// SIMATIC STEP 7 (V5.x) project examen2
// CPU: CPU 317-2 DP
// station: Hardware
// station: SIMATIC 300(1)
// station: P_ADR_BUS
// program: S7 Program(1)

SYMBOL_TABLE
"Prueba 1"	FB 1	FB 1
"Prueba 2"	FB 2	FB 2
"Prueba 3"	FB 3	FB 3
"Prueba 4"	FB 4	FB 4
"Prueba 5"	FB 5	FB 5
"Prueba 6"	FB 6	FB 6
"Prueba 8"	FB 8	FB 8
"Prueba 9"	FB 9	FB 9
"1HONGO"	I 0.0	BOOL
"1RESET"	I 0.1	BOOL
"1LOCAL"	I 0.2	BOOL
"1REMOTO"	I 0.3	BOOL
"1C_UNICO"	I 0.4	BOOL
"1C_CONTINUO"	I 0.5	BOOL
"1PARO"	I 0.6	BOOL
"1A0"	I 1.0	BOOL
"1A1"	I 1.1	BOOL
"1B0"	I 1.2	BOOL
"1B1"	I 1.3	BOOL
"2HONGO"	I 2.0	BOOL
"2RESET"	I 2.1	BOOL
"2LOCAL"	I 2.2	BOOL
"2REMOTO"	I 2.3	BOOL
"2C_UNICO"	I 2.4	BOOL
"2C_CONTINUO"	I 2.5	BOOL
"2PARO"	I 2.6	BOOL
"2A0"	I 3.0	BOOL
"2A1"	I 3.1	BOOL
"2B0"	I 3.2	BOOL
"2B1"	I 3.3	BOOL
"3HONGO"	I 4.0	BOOL
"3RESET"	I 4.1	BOOL
"3LOCAL"	I 4.2	BOOL
"3REMOTO"	I 4.3	BOOL
"3C_UNICO"	I 4.4	BOOL
"3C_CONTINUO"	I 4.5	BOOL
"3PARO"	I 4.6	BOOL
"3A0"	I 5.0	BOOL
"3A1"	I 5.1	BOOL
"3B0"	I 5.2	BOOL
"3B1"	I 5.3	BOOL
"3C0"	I 5.4	BOOL
"3C1"	I 5.5	BOOL
"4HONGO"	I 6.0	BOOL
"4RESET"	I 6.1	BOOL
"4LOCAL"	I 6.2	BOOL
"4REMOTO"	I 6.3	BOOL
"4C_UNICO"	I 6.4	BOOL
"4C_CONTINUO"	I 6.5	BOOL
"4PARO"	I 6.6	BOOL
"4C2"	I 6.7	BOOL
"4A0"	I 7.0	BOOL
"4A1"	I 7.1	BOOL
"4B0"	I 7.2	BOOL
"4B1"	I 7.3	BOOL
"4C0"	I 7.4	BOOL
"4C1"	I 7.5	BOOL
"4D0"	I 7.6	BOOL
"4D1"	I 7.7	BOOL
"5HONGO"	I 8.0	BOOL
"5RESET"	I 8.1	BOOL
"5LOCAL"	I 8.2	BOOL
"5REMOTO"	I 8.3	BOOL
"5C_UNICO"	I 8.4	BOOL
"5C_CONTINUO"	I 8.5	BOOL
"5PARO"	I 8.6	BOOL
"5A0"	I 9.0	BOOL
"5A1"	I 9.1	BOOL
"5B0"	I 9.2	BOOL
"5B1"	I 9.3	BOOL
"5C0"	I 9.4	BOOL
"5C1"	I 9.5	BOOL
"6HONGO"	I 10.0	BOOL
"6RESET"	I 10.1	BOOL
"6LOCAL"	I 10.2	BOOL
"6REMOTO"	I 10.3	BOOL
"6C_UNICO"	I 10.4	BOOL
"6C_CONTINUO"	I 10.5	BOOL
"6PARO"	I 10.6	BOOL
"6A0"	I 11.0	BOOL
"6A1"	I 11.1	BOOL
"6B0"	I 11.2	BOOL
"6B1"	I 11.3	BOOL
"6C0"	I 11.4	BOOL
"6C1"	I 11.5	BOOL
"6D0"	I 11.6	BOOL
"6D1"	I 11.7	BOOL
"8HONGO"	I 12.0	BOOL
"8RESET"	I 12.1	BOOL
"8LOCAL"	I 12.2	BOOL
"8REMOTO"	I 12.3	BOOL
"8C_UNICO"	I 12.4	BOOL
"8C_CONTINUO"	I 12.5	BOOL
"8PARO"	I 12.6	BOOL
"8A0"	I 13.0	BOOL
"8A1"	I 13.1	BOOL
"8B0"	I 13.2	BOOL
"8B1"	I 13.3	BOOL
"8C0"	I 13.4	BOOL
"8C1"	I 13.5	BOOL
"9HONGO"	I 14.0	BOOL
"9RESET"	I 14.1	BOOL
"9LOCAL"	I 14.2	BOOL
"9REMOTO"	I 14.3	BOOL
"9C_UNICO"	I 14.4	BOOL
"9C_CONTINUO"	I 14.5	BOOL
"9PARO"	I 14.6	BOOL
"9A1"	I 15.0	BOOL
"9A2"	I 15.1	BOOL
"9A3"	I 15.2	BOOL
"1Y1"	Q 0.0	BOOL
"1Y2"	Q 0.1	BOOL
"1Y3"	Q 0.2	BOOL
"1Y4"	Q 0.3	BOOL
"2Y1"	Q 1.0	BOOL
"2Y2"	Q 1.1	BOOL
"2Y3"	Q 1.2	BOOL
"2Y4"	Q 1.3	BOOL
"3Y1"	Q 2.0	BOOL
"3Y2"	Q 2.1	BOOL
"3Y3"	Q 2.2	BOOL
"3Y4"	Q 2.3	BOOL
"3Y5"	Q 2.4	BOOL
"3Y6"	Q 2.5	BOOL
"4Y1"	Q 3.0	BOOL
"4Y2"	Q 3.1	BOOL
"4Y3"	Q 3.2	BOOL
"4Y4"	Q 3.3	BOOL
"4Y5"	Q 3.4	BOOL
"4Y6"	Q 3.5	BOOL
"4Y7"	Q 3.6	BOOL
"4Y8"	Q 3.7	BOOL
"5Y1"	Q 4.0	BOOL
"5Y2"	Q 4.1	BOOL
"5Y3"	Q 4.2	BOOL
"5Y4"	Q 4.3	BOOL
"5Y5"	Q 4.4	BOOL
"5Y6"	Q 4.5	BOOL
"6Y1"	Q 5.0	BOOL
"6Y2"	Q 5.1	BOOL
"6Y3"	Q 5.2	BOOL
"6Y4"	Q 5.3	BOOL
"6Y5"	Q 5.4	BOOL
"6Y6"	Q 5.5	BOOL
"6Y7"	Q 5.6	BOOL
"6Y8"	Q 5.7	BOOL
"8Y1"	Q 6.0	BOOL
"8Y2"	Q 6.1	BOOL
"8Y3"	Q 6.2	BOOL
"8Y4"	Q 6.3	BOOL
"8Y5"	Q 6.4	BOOL
"8Y6"	Q 6.5	BOOL
"9Y1"	Q 7.0	BOOL
"9Y2"	Q 7.1	BOOL
END_SYMBOL_TABLE

FUNCTION_BLOCK "Prueba 1"	// FB 1
VERSION : 0.1
VAR
  K1 : BOOL ;
  KA : BOOL ;
  KB : BOOL ;
  K0 : BOOL ;
  K2 : BOOL ;
  K3 : BOOL ;
  K4 : BOOL ;
  K5 : BOOL ;
  K6 : BOOL ;
  K7 : BOOL ;
  K8 : BOOL ;
  KT8 : BOOL ;
  K9 : BOOL ;
END_VAR
BEGIN
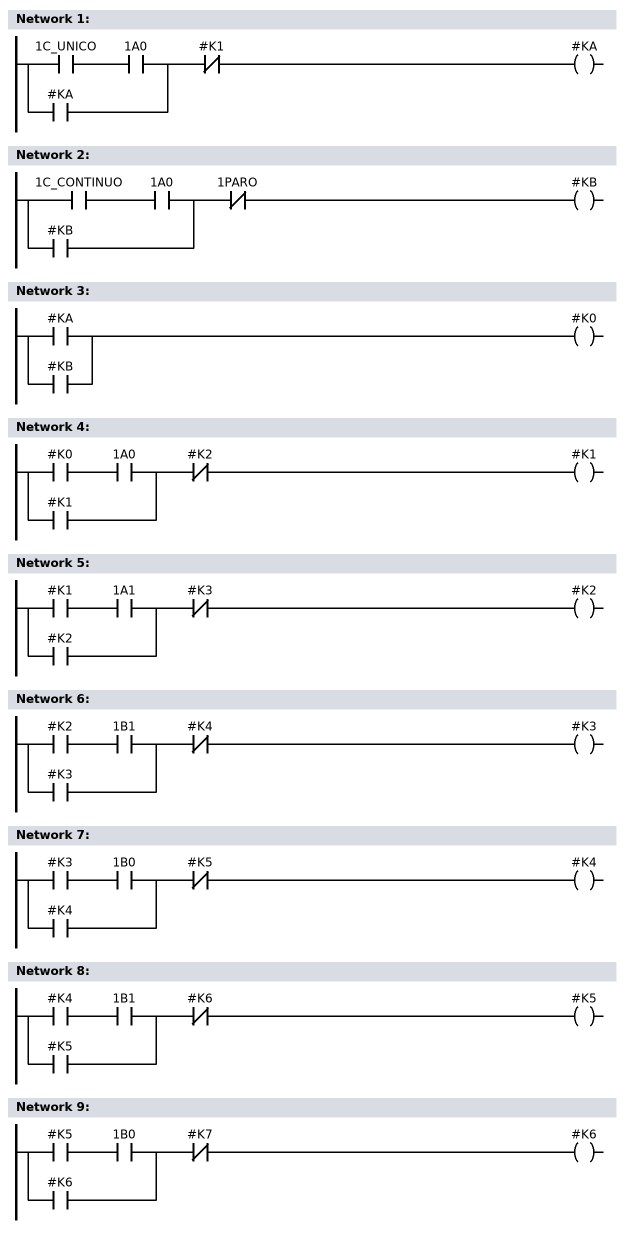
NETWORK
TITLE =
      A(;
      A     "1C_UNICO";
      A     "1A0";
      O     #KA;
      );
      AN    #K1;
      =     #KA;
NETWORK
TITLE =
      A(;
      A     "1C_CONTINUO";
      A     "1A0";
      O     #KB;
      );
      AN    "1PARO";
      =     #KB;
NETWORK
TITLE =
      O     #KA;
      O     #KB;
      =     #K0;
NETWORK
TITLE =
      A(;
      A     #K0;
      A     "1A0";
      O     #K1;
      );
      AN    #K2;
      =     #K1;
NETWORK
TITLE =
      A(;
      A     #K1;
      A     "1A1";
      O     #K2;
      );
      AN    #K3;
      =     #K2;
NETWORK
TITLE =
      A(;
      A     #K2;
      A     "1B1";
      O     #K3;
      );
      AN    #K4;
      =     #K3;
NETWORK
TITLE =
      A(;
      A     #K3;
      A     "1B0";
      O     #K4;
      );
      AN    #K5;
      =     #K4;
NETWORK
TITLE =
      A(;
      A     #K4;
      A     "1B1";
      O     #K5;
      );
      AN    #K6;
      =     #K5;
NETWORK
TITLE =
      A(;
      A     #K5;
      A     "1B0";
      O     #K6;
      );
      AN    #K7;
      =     #K6;
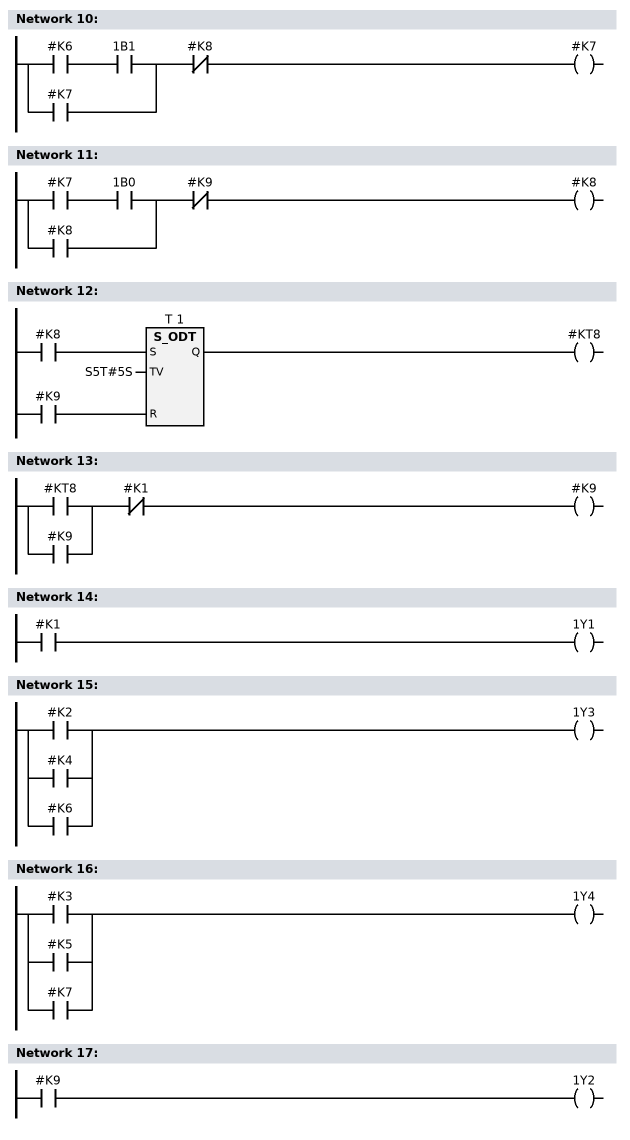
NETWORK
TITLE =
      A(;
      A     #K6;
      A     "1B1";
      O     #K7;
      );
      AN    #K8;
      =     #K7;
NETWORK
TITLE =
      A(;
      A     #K7;
      A     "1B0";
      O     #K8;
      );
      AN    #K9;
      =     #K8;
NETWORK
TITLE =
      A     #K8;
      L     S5T#5S;
      SD    T 1;
      A     #K9;
      R     T 1;
      NOP   0;
      NOP   0;
      A     T 1;
      =     #KT8;
NETWORK
TITLE =
      A(;
      O     #KT8;
      O     #K9;
      );
      AN    #K1;
      =     #K9;
NETWORK
TITLE =
      A     #K1;
      =     "1Y1";
NETWORK
TITLE =
      O     #K2;
      O     #K4;
      O     #K6;
      =     "1Y3";
NETWORK
TITLE =
      O     #K3;
      O     #K5;
      O     #K7;
      =     "1Y4";
NETWORK
TITLE =
      A     #K9;
      =     "1Y2";
END_FUNCTION_BLOCK

FUNCTION_BLOCK "Prueba 2"	// FB 2
VERSION : 0.1
VAR
  K0 : BOOL ;
  K1 : BOOL ;
  K2 : BOOL ;
  K3 : BOOL ;
  K4 : BOOL ;
  K5 : BOOL ;
  K6 : BOOL ;
  K7 : BOOL ;
  K8 : BOOL ;
  KT : BOOL ;
  KA : BOOL ;
  KB : BOOL ;
  kt2 : BOOL ;
END_VAR
BEGIN
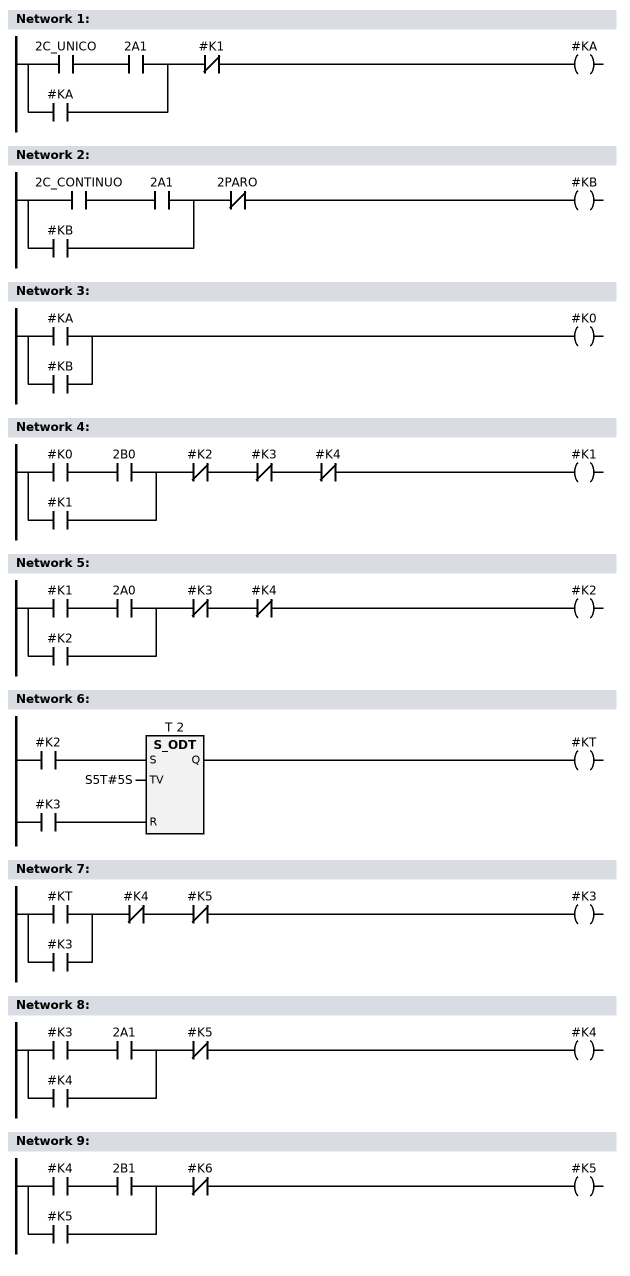
NETWORK
TITLE =
      A(;
      A     "2C_UNICO";
      A     "2A1";
      O     #KA;
      );
      AN    #K1;
      =     #KA;
NETWORK
TITLE =
      A(;
      A     "2C_CONTINUO";
      A     "2A1";
      O     #KB;
      );
      AN    "2PARO";
      =     #KB;
NETWORK
TITLE =
      O     #KA;
      O     #KB;
      =     #K0;
NETWORK
TITLE =
      A(;
      A     #K0;
      A     "2B0";
      O     #K1;
      );
      AN    #K2;
      AN    #K3;
      AN    #K4;
      =     #K1;
NETWORK
TITLE =
      A(;
      A     #K1;
      A     "2A0";
      O     #K2;
      );
      AN    #K3;
      AN    #K4;
      =     #K2;
NETWORK
TITLE =
      A     #K2;
      L     S5T#5S;
      SD    T 2;
      A     #K3;
      R     T 2;
      NOP   0;
      NOP   0;
      A     T 2;
      =     #KT;
NETWORK
TITLE =
      A(;
      O     #KT;
      O     #K3;
      );
      AN    #K4;
      AN    #K5;
      =     #K3;
NETWORK
TITLE =
      A(;
      A     #K3;
      A     "2A1";
      O     #K4;
      );
      AN    #K5;
      =     #K4;
NETWORK
TITLE =
      A(;
      A     #K4;
      A     "2B1";
      O     #K5;
      );
      AN    #K6;
      =     #K5;
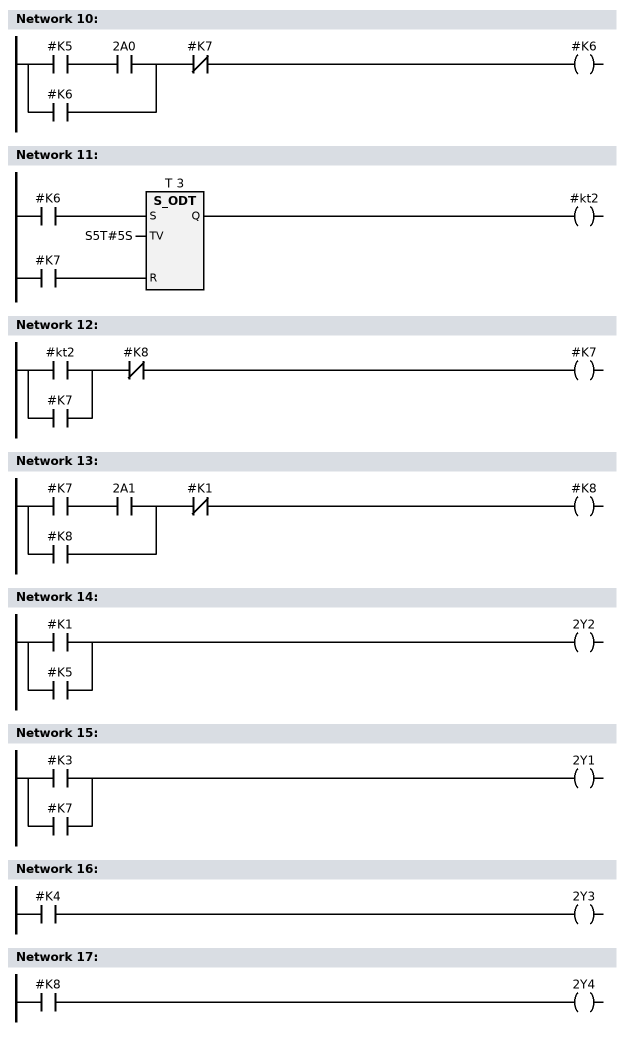
NETWORK
TITLE =
      A(;
      A     #K5;
      A     "2A0";
      O     #K6;
      );
      AN    #K7;
      =     #K6;
NETWORK
TITLE =
      A     #K6;
      L     S5T#5S;
      SD    T 3;
      A     #K7;
      R     T 3;
      NOP   0;
      NOP   0;
      A     T 3;
      =     #kt2;
NETWORK
TITLE =
      A(;
      O     #kt2;
      O     #K7;
      );
      AN    #K8;
      =     #K7;
NETWORK
TITLE =
      A(;
      A     #K7;
      A     "2A1";
      O     #K8;
      );
      AN    #K1;
      =     #K8;
NETWORK
TITLE =
      O     #K1;
      O     #K5;
      =     "2Y2";
NETWORK
TITLE =
      O     #K3;
      O     #K7;
      =     "2Y1";
NETWORK
TITLE =
      A     #K4;
      =     "2Y3";
NETWORK
TITLE =
      A     #K8;
      =     "2Y4";
END_FUNCTION_BLOCK

FUNCTION_BLOCK "Prueba 3"	// FB 3
VERSION : 0.1
VAR
  KA : BOOL ;
  KB : BOOL ;
  K0 : BOOL ;
  K1 : BOOL ;
  K2 : BOOL ;
  K3 : BOOL ;
  K4 : BOOL ;
  K5 : BOOL ;
  K6 : BOOL ;
  K7 : BOOL ;
END_VAR
BEGIN
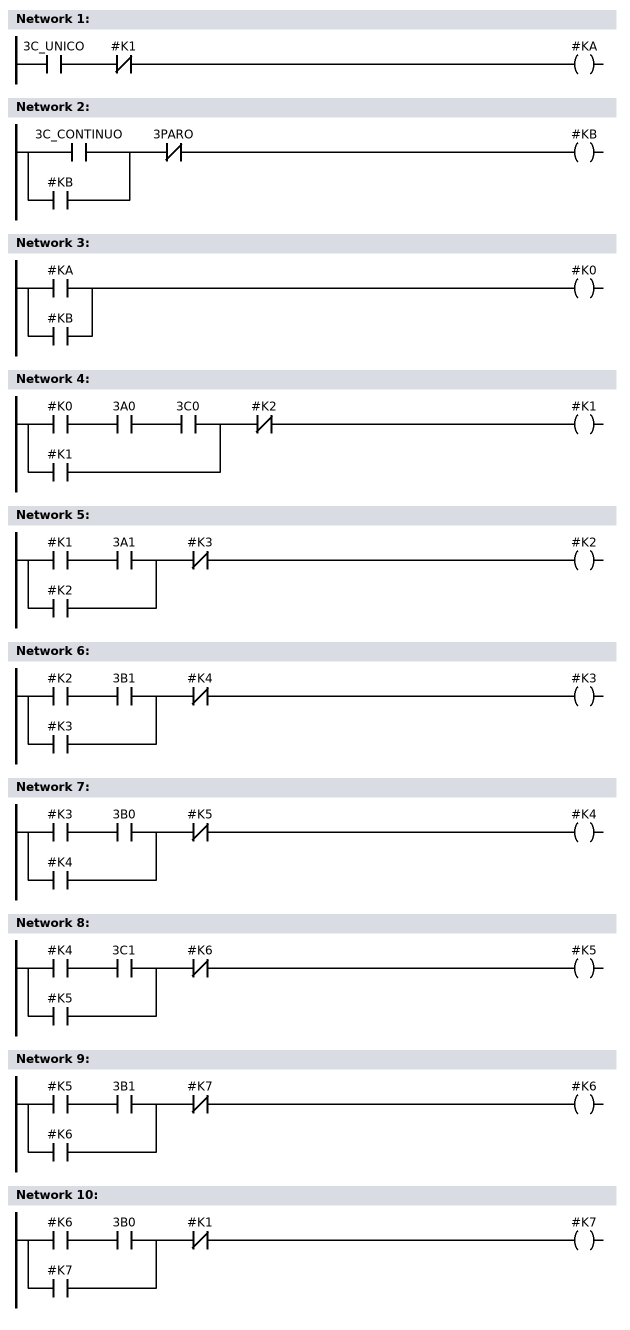
NETWORK
TITLE =
      A     "3C_UNICO";
      AN    #K1;
      =     #KA;
NETWORK
TITLE =
      A(;
      O     "3C_CONTINUO";
      O     #KB;
      );
      AN    "3PARO";
      =     #KB;
NETWORK
TITLE =
      O     #KA;
      O     #KB;
      =     #K0;
NETWORK
TITLE =
      A(;
      A     #K0;
      A     "3A0";
      A     "3C0";
      O     #K1;
      );
      AN    #K2;
      =     #K1;
NETWORK
TITLE =
      A(;
      A     #K1;
      A     "3A1";
      O     #K2;
      );
      AN    #K3;
      =     #K2;
NETWORK
TITLE =
      A(;
      A     #K2;
      A     "3B1";
      O     #K3;
      );
      AN    #K4;
      =     #K3;
NETWORK
TITLE =
      A(;
      A     #K3;
      A     "3B0";
      O     #K4;
      );
      AN    #K5;
      =     #K4;
NETWORK
TITLE =
      A(;
      A     #K4;
      A     "3C1";
      O     #K5;
      );
      AN    #K6;
      =     #K5;
NETWORK
TITLE =
      A(;
      A     #K5;
      A     "3B1";
      O     #K6;
      );
      AN    #K7;
      =     #K6;
NETWORK
TITLE =
      A(;
      A     #K6;
      A     "3B0";
      O     #K7;
      );
      AN    #K1;
      =     #K7;
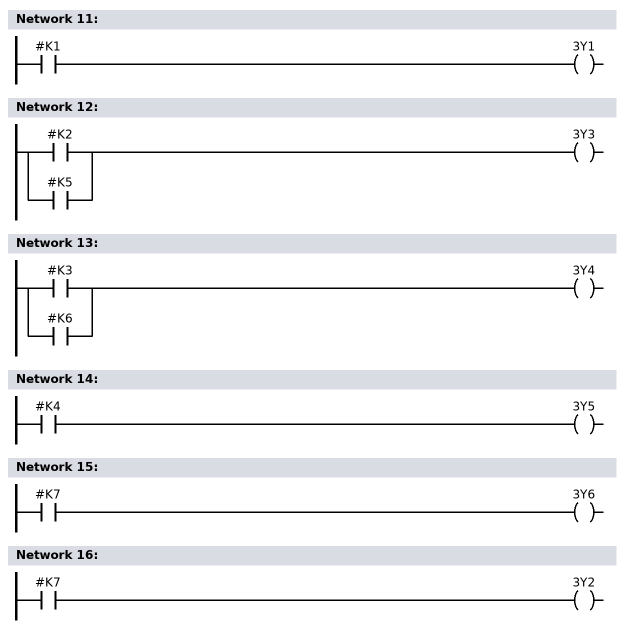
NETWORK
TITLE =
      A     #K1;
      =     "3Y1";
NETWORK
TITLE =
      O     #K2;
      O     #K5;
      =     "3Y3";
NETWORK
TITLE =
      O     #K3;
      O     #K6;
      =     "3Y4";
NETWORK
TITLE =
      A     #K4;
      =     "3Y5";
NETWORK
TITLE =
      A     #K7;
      =     "3Y6";
NETWORK
TITLE =
      A     #K7;
      =     "3Y2";
END_FUNCTION_BLOCK

FUNCTION_BLOCK "Prueba 4"	// FB 4
TITLE = Prueba 4
VERSION : 0.1
VAR
  KA : BOOL ;
  KB : BOOL ;
  K0 : BOOL ;
  K1 : BOOL ;
  K2 : BOOL ;
  K3 : BOOL ;
  K4 : BOOL ;
  K5 : BOOL ;
  K6 : BOOL ;
  K7 : BOOL ;
  K8 : BOOL ;
  K9 : BOOL ;
  KT : BOOL ;
END_VAR
BEGIN
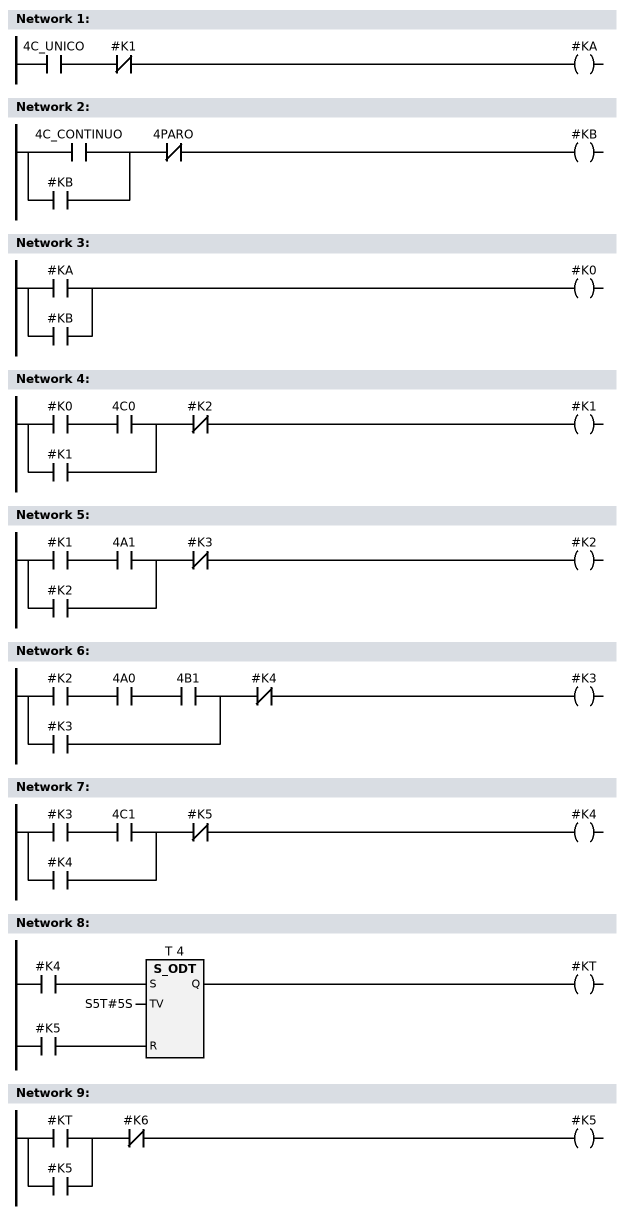
NETWORK
TITLE =
      A     "4C_UNICO";
      AN    #K1;
      =     #KA;
NETWORK
TITLE =
      A(;
      O     "4C_CONTINUO";
      O     #KB;
      );
      AN    "4PARO";
      =     #KB;
NETWORK
TITLE =
      O     #KA;
      O     #KB;
      =     #K0;
NETWORK
TITLE =
      A(;
      A     #K0;
      A     "4C0";
      O     #K1;
      );
      AN    #K2;
      =     #K1;
NETWORK
TITLE =
      A(;
      A     #K1;
      A     "4A1";
      O     #K2;
      );
      AN    #K3;
      =     #K2;
NETWORK
TITLE =
      A(;
      A     #K2;
      A     "4A0";
      A     "4B1";
      O     #K3;
      );
      AN    #K4;
      =     #K3;
NETWORK
TITLE =
      A(;
      A     #K3;
      A     "4C1";
      O     #K4;
      );
      AN    #K5;
      =     #K4;
NETWORK
TITLE =
      A     #K4;
      L     S5T#5S;
      SD    T 4;
      A     #K5;
      R     T 4;
      NOP   0;
      NOP   0;
      A     T 4;
      =     #KT;
NETWORK
TITLE =
      A(;
      O     #KT;
      O     #K5;
      );
      AN    #K6;
      =     #K5;
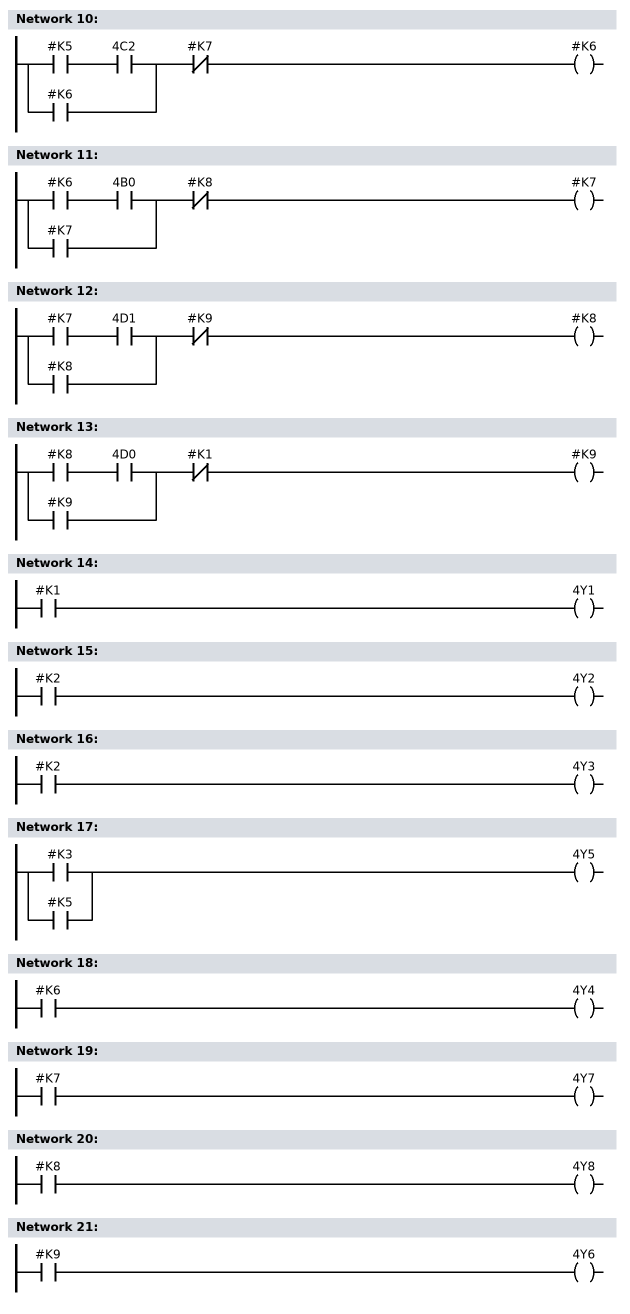
NETWORK
TITLE =
      A(;
      A     #K5;
      A     "4C2";
      O     #K6;
      );
      AN    #K7;
      =     #K6;
NETWORK
TITLE =
      A(;
      A     #K6;
      A     "4B0";
      O     #K7;
      );
      AN    #K8;
      =     #K7;
NETWORK
TITLE =
      A(;
      A     #K7;
      A     "4D1";
      O     #K8;
      );
      AN    #K9;
      =     #K8;
NETWORK
TITLE =
      A(;
      A     #K8;
      A     "4D0";
      O     #K9;
      );
      AN    #K1;
      =     #K9;
NETWORK
TITLE =
      A     #K1;
      =     "4Y1";
NETWORK
TITLE =
      A     #K2;
      =     "4Y2";
NETWORK
TITLE =
      A     #K2;
      =     "4Y3";
NETWORK
TITLE =
      O     #K3;
      O     #K5;
      =     "4Y5";
NETWORK
TITLE =
      A     #K6;
      =     "4Y4";
NETWORK
TITLE =
      A     #K7;
      =     "4Y7";
NETWORK
TITLE =
      A     #K8;
      =     "4Y8";
NETWORK
TITLE =
      A     #K9;
      =     "4Y6";
END_FUNCTION_BLOCK

FUNCTION_BLOCK "Prueba 5"	// FB 5
VERSION : 0.1
VAR
  KA : BOOL ;
  KB : BOOL ;
  K0 : BOOL ;
  K1 : BOOL ;
  K2 : BOOL ;
  K3 : BOOL ;
  K4 : BOOL ;
  K5 : BOOL ;
  K6 : BOOL ;
  K7 : BOOL ;
  K8 : BOOL ;
  K9 : BOOL ;
END_VAR
BEGIN
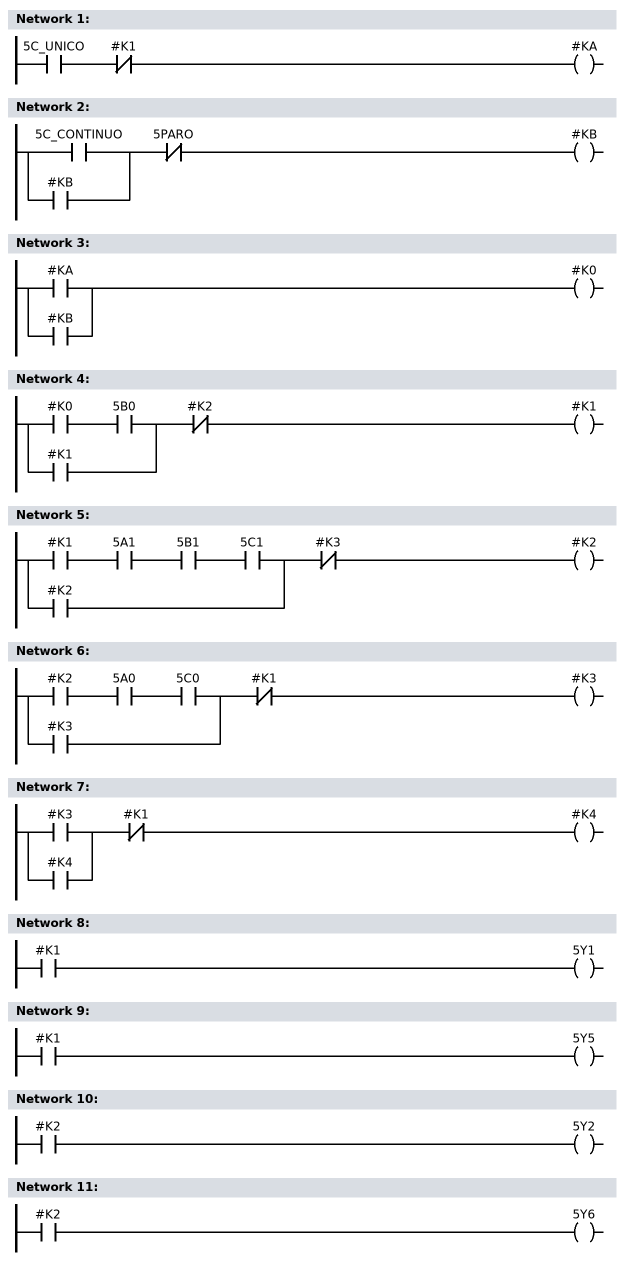
NETWORK
TITLE =
      A     "5C_UNICO";
      AN    #K1;
      =     #KA;
NETWORK
TITLE =
      A(;
      O     "5C_CONTINUO";
      O     #KB;
      );
      AN    "5PARO";
      =     #KB;
NETWORK
TITLE =
      O     #KA;
      O     #KB;
      =     #K0;
NETWORK
TITLE =
      A(;
      A     #K0;
      A     "5B0";
      O     #K1;
      );
      AN    #K2;
      =     #K1;
NETWORK
TITLE =
      A(;
      A     #K1;
      A     "5A1";
      A     "5B1";
      A     "5C1";
      O     #K2;
      );
      AN    #K3;
      =     #K2;
NETWORK
TITLE =
      A(;
      A     #K2;
      A     "5A0";
      A     "5C0";
      O     #K3;
      );
      AN    #K1;
      =     #K3;
NETWORK
TITLE =
      A(;
      O     #K3;
      O     #K4;
      );
      AN    #K1;
      =     #K4;
NETWORK
TITLE =
      A     #K1;
      =     "5Y1";
NETWORK
TITLE =
      A     #K1;
      =     "5Y5";
NETWORK
TITLE =
      A     #K2;
      =     "5Y2";
NETWORK
TITLE =
      A     #K2;
      =     "5Y6";
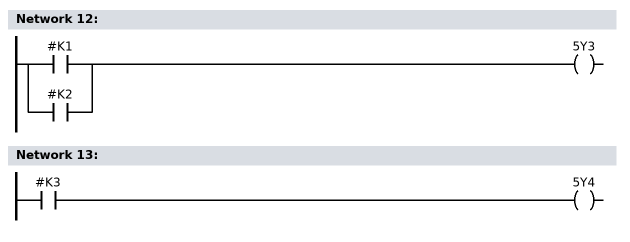
NETWORK
TITLE =
      O     #K1;
      O     #K2;
      =     "5Y3";
NETWORK
TITLE =
      A     #K3;
      =     "5Y4";
END_FUNCTION_BLOCK

FUNCTION_BLOCK "Prueba 6"	// FB 6
VERSION : 0.1
VAR
  KA : BOOL ;
  KB : BOOL ;
  K0 : BOOL ;
  K1 : BOOL ;
  K2 : BOOL ;
  K3 : BOOL ;
  K4 : BOOL ;
  K5 : BOOL ;
  K6 : BOOL ;
  K7 : BOOL ;
  K8 : BOOL ;
  K9 : BOOL ;
END_VAR
BEGIN
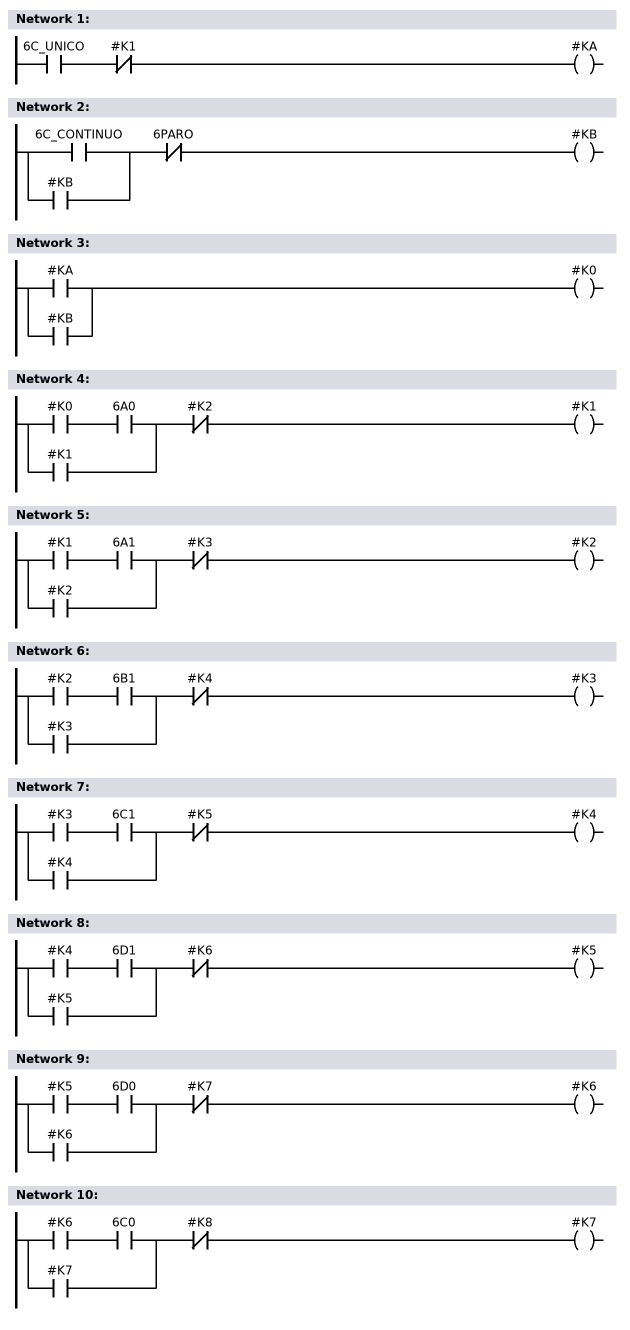
NETWORK
TITLE =
      A     "6C_UNICO";
      AN    #K1;
      =     #KA;
NETWORK
TITLE =
      A(;
      O     "6C_CONTINUO";
      O     #KB;
      );
      AN    "6PARO";
      =     #KB;
NETWORK
TITLE =
      O     #KA;
      O     #KB;
      =     #K0;
NETWORK
TITLE =
      A(;
      A     #K0;
      A     "6A0";
      O     #K1;
      );
      AN    #K2;
      =     #K1;
NETWORK
TITLE =
      A(;
      A     #K1;
      A     "6A1";
      O     #K2;
      );
      AN    #K3;
      =     #K2;
NETWORK
TITLE =
      A(;
      A     #K2;
      A     "6B1";
      O     #K3;
      );
      AN    #K4;
      =     #K3;
NETWORK
TITLE =
      A(;
      A     #K3;
      A     "6C1";
      O     #K4;
      );
      AN    #K5;
      =     #K4;
NETWORK
TITLE =
      A(;
      A     #K4;
      A     "6D1";
      O     #K5;
      );
      AN    #K6;
      =     #K5;
NETWORK
TITLE =
      A(;
      A     #K5;
      A     "6D0";
      O     #K6;
      );
      AN    #K7;
      =     #K6;
NETWORK
TITLE =
      A(;
      A     #K6;
      A     "6C0";
      O     #K7;
      );
      AN    #K8;
      =     #K7;
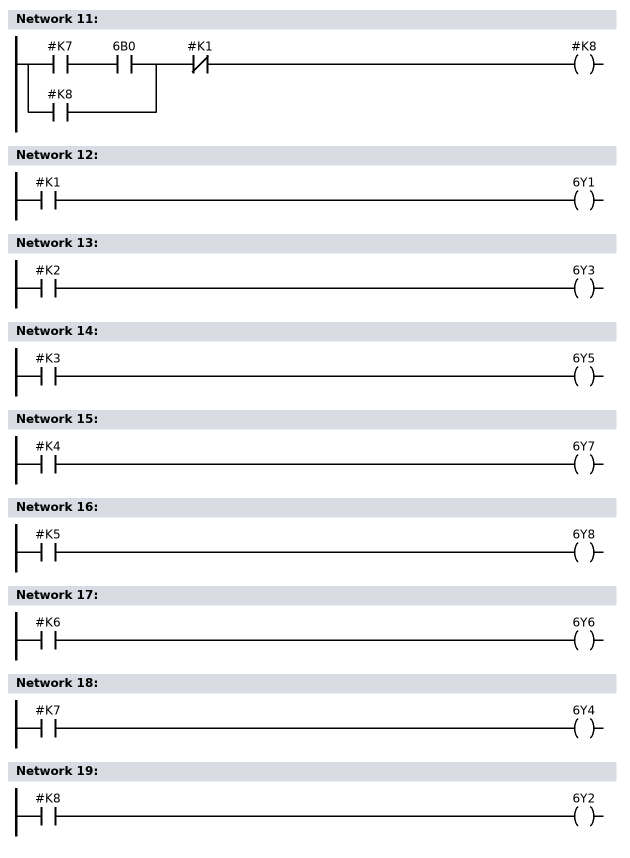
NETWORK
TITLE =
      A(;
      A     #K7;
      A     "6B0";
      O     #K8;
      );
      AN    #K1;
      =     #K8;
NETWORK
TITLE =
      A     #K1;
      =     "6Y1";
NETWORK
TITLE =
      A     #K2;
      =     "6Y3";
NETWORK
TITLE =
      A     #K3;
      =     "6Y5";
NETWORK
TITLE =
      A     #K4;
      =     "6Y7";
NETWORK
TITLE =
      A     #K5;
      =     "6Y8";
NETWORK
TITLE =
      A     #K6;
      =     "6Y6";
NETWORK
TITLE =
      A     #K7;
      =     "6Y4";
NETWORK
TITLE =
      A     #K8;
      =     "6Y2";
END_FUNCTION_BLOCK

FUNCTION_BLOCK "Prueba 8"	// FB 8
VERSION : 0.1
VAR
  KA : BOOL ;
  KB : BOOL ;
  K0 : BOOL ;
  K1 : BOOL ;
  K2 : BOOL ;
  K3 : BOOL ;
  K4 : BOOL ;
  K5 : BOOL ;
  K6 : BOOL ;
  K7 : BOOL ;
  K8 : BOOL ;
  K9 : BOOL ;
END_VAR
BEGIN
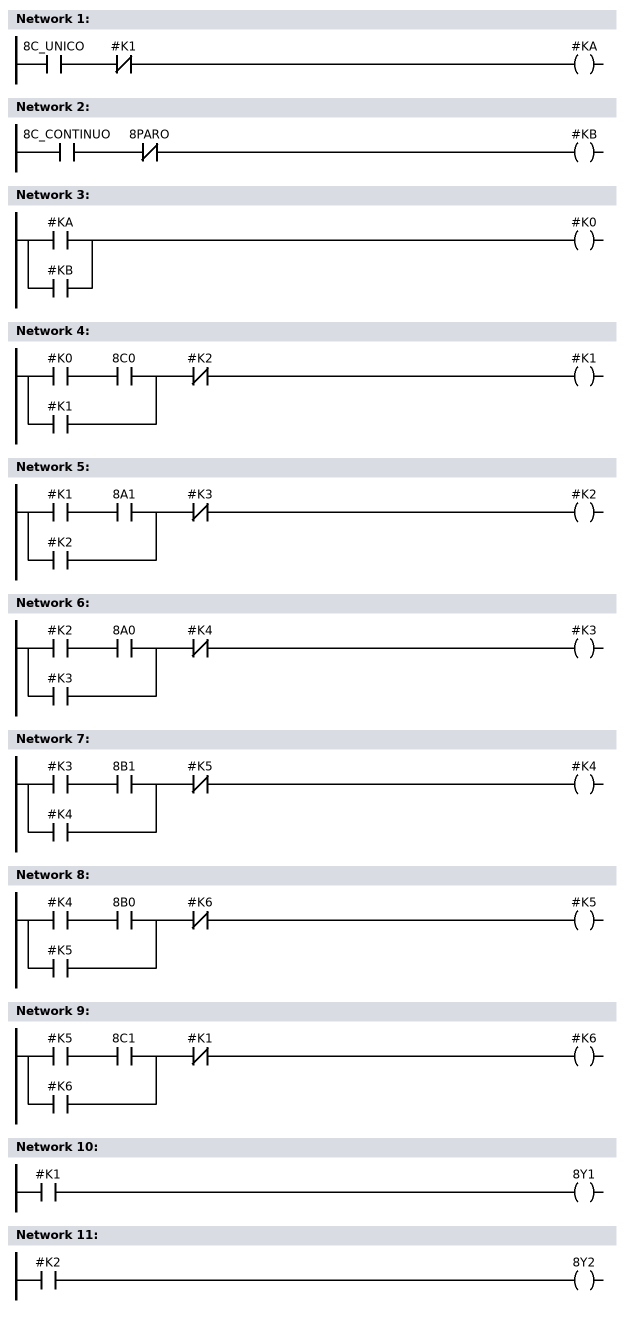
NETWORK
TITLE =
      A     "8C_UNICO";
      AN    #K1;
      =     #KA;
NETWORK
TITLE =
      A     "8C_CONTINUO";
      AN    "8PARO";
      =     #KB;
NETWORK
TITLE =
      O     #KA;
      O     #KB;
      =     #K0;
NETWORK
TITLE =
      A(;
      A     #K0;
      A     "8C0";
      O     #K1;
      );
      AN    #K2;
      =     #K1;
NETWORK
TITLE =
      A(;
      A     #K1;
      A     "8A1";
      O     #K2;
      );
      AN    #K3;
      =     #K2;
NETWORK
TITLE =
      A(;
      A     #K2;
      A     "8A0";
      O     #K3;
      );
      AN    #K4;
      =     #K3;
NETWORK
TITLE =
      A(;
      A     #K3;
      A     "8B1";
      O     #K4;
      );
      AN    #K5;
      =     #K4;
NETWORK
TITLE =
      A(;
      A     #K4;
      A     "8B0";
      O     #K5;
      );
      AN    #K6;
      =     #K5;
NETWORK
TITLE =
      A(;
      A     #K5;
      A     "8C1";
      O     #K6;
      );
      AN    #K1;
      =     #K6;
NETWORK
TITLE =
      A     #K1;
      =     "8Y1";
NETWORK
TITLE =
      A     #K2;
      =     "8Y2";
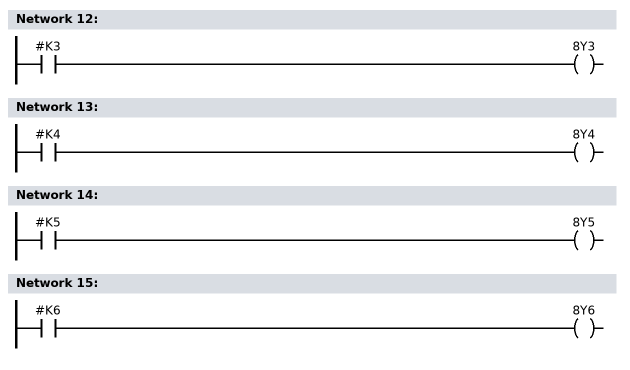
NETWORK
TITLE =
      A     #K3;
      =     "8Y3";
NETWORK
TITLE =
      A     #K4;
      =     "8Y4";
NETWORK
TITLE =
      A     #K5;
      =     "8Y5";
NETWORK
TITLE =
      A     #K6;
      =     "8Y6";
END_FUNCTION_BLOCK

FUNCTION_BLOCK "Prueba 9"	// FB 9
VERSION : 0.1
VAR
  KA : BOOL ;
  KB : BOOL ;
  K0 : BOOL ;
  K1 : BOOL ;
  K2 : BOOL ;
  K3 : BOOL ;
  K4 : BOOL ;
END_VAR
BEGIN
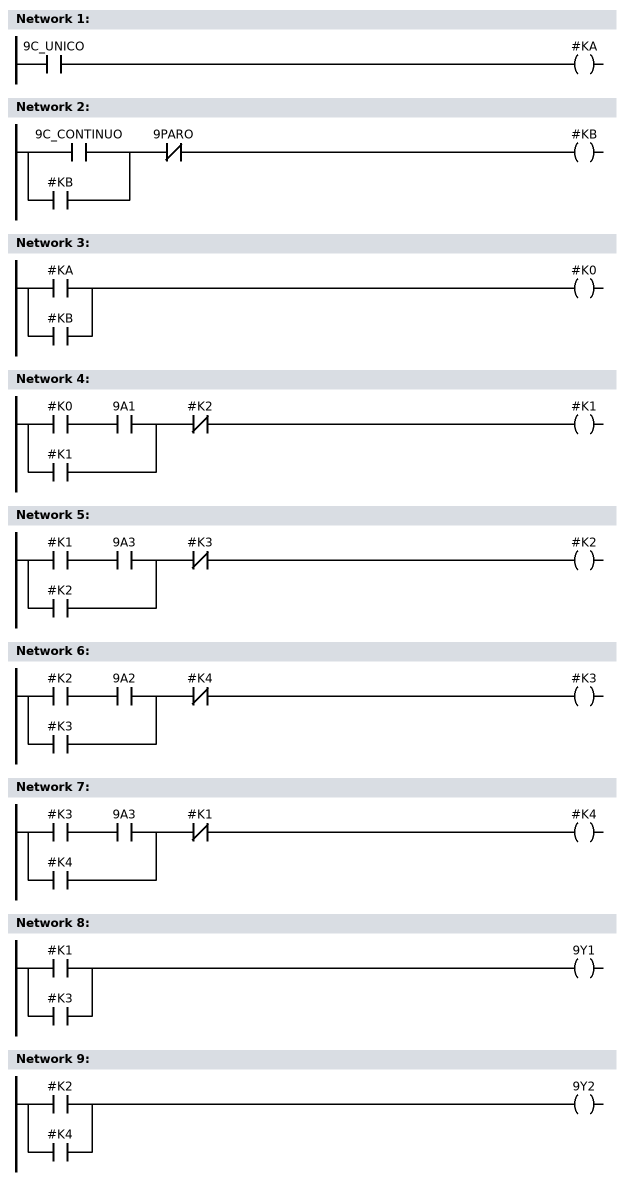
NETWORK
TITLE =
      A     "9C_UNICO";
      =     #KA;
NETWORK
TITLE =
      A(;
      O     "9C_CONTINUO";
      O     #KB;
      );
      AN    "9PARO";
      =     #KB;
NETWORK
TITLE =
      O     #KA;
      O     #KB;
      =     #K0;
NETWORK
TITLE =
      A(;
      A     #K0;
      A     "9A1";
      O     #K1;
      );
      AN    #K2;
      =     #K1;
NETWORK
TITLE =
      A(;
      A     #K1;
      A     "9A3";
      O     #K2;
      );
      AN    #K3;
      =     #K2;
NETWORK
TITLE =
      A(;
      A     #K2;
      A     "9A2";
      O     #K3;
      );
      AN    #K4;
      =     #K3;
NETWORK
TITLE =
      A(;
      A     #K3;
      A     "9A3";
      O     #K4;
      );
      AN    #K1;
      =     #K4;
NETWORK
TITLE =
      O     #K1;
      O     #K3;
      =     "9Y1";
NETWORK
TITLE =
      O     #K2;
      O     #K4;
      =     "9Y2";
END_FUNCTION_BLOCK

DATA_BLOCK DB 1
VERSION : 0.0
"Prueba 1"
BEGIN
END_DATA_BLOCK

DATA_BLOCK DB 2
VERSION : 0.0
"Prueba 2"
BEGIN
END_DATA_BLOCK

DATA_BLOCK DB 3
VERSION : 0.0
"Prueba 3"
BEGIN
END_DATA_BLOCK

DATA_BLOCK DB 4
VERSION : 0.0
"Prueba 4"
BEGIN
END_DATA_BLOCK

DATA_BLOCK DB 5
VERSION : 0.0
"Prueba 5"
BEGIN
END_DATA_BLOCK

DATA_BLOCK DB 6
VERSION : 0.0
"Prueba 6"
BEGIN
END_DATA_BLOCK

DATA_BLOCK DB 8
VERSION : 0.0
"Prueba 8"
BEGIN
END_DATA_BLOCK

DATA_BLOCK DB 9
VERSION : 0.0
"Prueba 9"
BEGIN
END_DATA_BLOCK

ORGANIZATION_BLOCK OB 1
TITLE = "Main Program Sweep (Cycle)"
VERSION : 0.1
VAR_TEMP
  OB1_EV_CLASS : BYTE ;	//Bits 0-3 = 1 (Coming event), Bits 4-7 = 1 (Event class 1)
  OB1_SCAN_1 : BYTE ;	//1 (Cold restart scan 1 of OB 1), 3 (Scan 2-n of OB 1)
  OB1_PRIORITY : BYTE ;	//Priority of OB Execution
  OB1_OB_NUMBR : BYTE ;	//1 (Organization block 1, OB1)
  OB1_RESERVED_1 : BYTE ;	//Reserved for system
  OB1_RESERVED_2 : BYTE ;	//Reserved for system
  OB1_PREV_CYCLE : INT ;	//Cycle time of previous OB1 scan (milliseconds)
  OB1_MIN_CYCLE : INT ;	//Minimum cycle time of OB1 (milliseconds)
  OB1_MAX_CYCLE : INT ;	//Maximum cycle time of OB1 (milliseconds)
  OB1_DATE_TIME : DATE_AND_TIME ;	//Date and time OB1 started
END_VAR
BEGIN
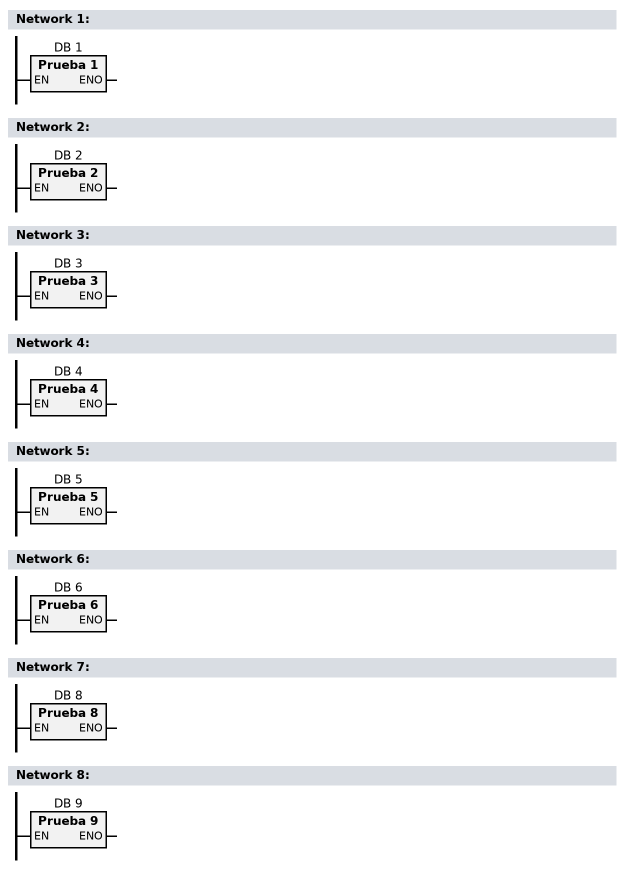
NETWORK
TITLE =
      CALL  "Prueba 1" , DB 1;
      NOP   0;
NETWORK
TITLE =
      CALL  "Prueba 2" , DB 2;
      NOP   0;
NETWORK
TITLE =
      CALL  "Prueba 3" , DB 3;
      NOP   0;
NETWORK
TITLE =
      CALL  "Prueba 4" , DB 4;
      NOP   0;
NETWORK
TITLE =
      CALL  "Prueba 5" , DB 5;
      NOP   0;
NETWORK
TITLE =
      CALL  "Prueba 6" , DB 6;
      NOP   0;
NETWORK
TITLE =
      CALL  "Prueba 8" , DB 8;
      NOP   0;
NETWORK
TITLE =
      CALL  "Prueba 9" , DB 9;
      NOP   0;
END_ORGANIZATION_BLOCK
